# B&R Automation Studio project Code_für_SPS
Automation Studio 4.9

## Configuration Config1

CPU X20CP1382, AutomationRuntime B4.63, Build 4.1.2, Vc V4.62.0

### Task classes (Cpu.sw)
```
Cyclic#4:
  Program1 <- Program1.prg
Binaries: udbdef, mvLoader, FWRules, TCData, ashwac, arconfig, asfw, ashwd, iomap, User, Role, sysconf
Libraries: sys_lib, AsBrStr, runtime, Library, standard, fileio, astime, asieccon
```

### Hardware
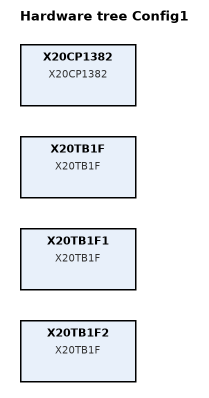
```
X20CP1382 : X20CP1382 v1.14.0.0  [X1 -> X1.SL; X2 -> X2.SL; X3 -> X3.SL]
  Module X1 (Type=X1, Virtual=true, Version=1.14.0.0)
    Connection (Connector=SS1, TargetModule=X20TB1F, TargetConnector=SS)
    Connection (Connector=SL, TargetModule=X20CP1382, TargetConnector=X1)
  Module X2 (Type=X2, Virtual=true, Version=1.14.0.0)
    Connection (Connector=SS1, TargetModule=X20TB1F1, TargetConnector=SS)
    Connection (Connector=SL, TargetModule=X20CP1382, TargetConnector=X2)
  Module X3 (Type=X3, Virtual=true, Version=1.14.0.0)
    Connection (Connector=SS1, TargetModule=X20TB1F2, TargetConnector=SS)
    Connection (Connector=SL, TargetModule=X20CP1382, TargetConnector=X3)
  Connector IF2:
    ActivateDevice = 1
    HostName = x20cp1382
    Mode = Manual
    InternetAddress = 192.168.1.10
    SubnetMask = 255.255.255.0
    InaNodeNumber = 0
  Connector IF3:
    DNAConfiguration = manual
  ConfigurationID = Cocktailmaschine_Config1
  ActivateOpcUa = 1
  OpcUaInformationModels_PV_Version = 1
X20TB1F : X20TB1F v1.0.0.0
X20TB1F1 : X20TB1F v1.0.0.0
X20TB1F2 : X20TB1F v1.0.0.0
```

### IoMap.iom - X20CP1382/IoMap.iom
```iecst
VAR_CONFIG
	::Program1:OutVentil2 AT %QX."X3".DigitalOutput02;
	::Program1:InLichtschranke AT %IX."X2".DigitalInput01;
	::Program1:OutVentil1 AT %QX."X3".DigitalOutput01;
	::Program1:OutVentil3 AT %QX."X3".DigitalOutput03;
	::Program1:OutVentil4 AT %QX."X3".DigitalOutput04;
	::Program1:OutVentil5 AT %QX."X3".DigitalOutput05;
	::Program1:OutVentil6 AT %QX."X3".DigitalOutput06;
	::Program1:OutVentil7 AT %QX."X3".DigitalOutput07;
	::Program1:OutVentil8 AT %QX."X3".DigitalOutput08;
	::Program1:OutPumpe AT %QX."X3".DigitalOutput09;
	::Program1:OutMotorEis AT %QX."X3".DigitalOutput10;
	::Program1:OutLampeGruen AT %QX."X3".DigitalOutput11;
	::Program1:OutLampeRot AT %QX."X3".DigitalOutput12;
	::Program1:InEndlageMotor AT %IX."X2".DigitalInput02;
	::Program1:InEndlageMotor2 AT %IX."X2".DigitalInput03;
	::Program1:InAnalogWaage AT %IW."X1".AnalogInput02;
END_VAR
```

## Logical view

Binary libraries used (declarations not repeated): operator, runtime, astime, AsIecCon, sys_lib, AsBrStr, standard

### Library Logical/Library (IEC)

#### Library.fun - Exported functions and function blocks
```iecst
{REDUND_ERROR} FUNCTION setOutputs : BOOL (*TODO: Add your comment here*) (*$GROUP=User,$CAT=User,$GROUPICON=User.png,$CATICON=User.png*)
	VAR_INPUT
		ventil1 : BOOL;
		ventil2 : BOOL;
		ventil3 : BOOL;
		ventil4 : BOOL;
		ventil5 : BOOL;
		ventil6 : BOOL;
		ventil7 : BOOL;
		ventil8 : BOOL;
		rot : BOOL;
		gruen : BOOL;
		pumpe : BOOL;
		motor : BOOL;
	END_VAR
END_FUNCTION
```

#### setOutputs.ab
```automation-basic
(* TODO: Add your comment here *)
FUNCTION setOutputs
	//OutVentil1 := ventil1;
	//OutVentil2 := ventil2;
	//OutVentil3 := ventil3;
	//OutVentil4 := ventil4;
	//OutVentil5 := ventil5;
	//OutVentil6 := ventil6;
	//OutVentil7 := ventil7;
	//OutVentil8 := ventil8;
	//OutLampeRot := rot;
	//OutLampeGruen := gruen;
	//OutPumpe := pumpe;
	//OutMotorEis := motor;
END_FUNCTION
```

### Package Logical/Libraries - Globale Bibliotheken

- Visualisation Logical/mappView (not shown)

### Program Logical/Program (IEC)

#### Cyclic.st - Cyclic code
```iecst
PROGRAM _CYCLIC
	IF Zustand = TRUE THEN
		//Hier kommt der Befehl zum Anzeigen dert Startseite hin
		OutVentil1 := FALSE;OutVentil2 := FALSE;OutVentil3 := FALSE;OutVentil4 := FALSE;OutVentil5 := FALSE;OutVentil6 := FALSE;
		OutVentil7 := FALSE;OutVentil8 := FALSE;OutLampeRot := FALSE;OutLampeGruen := FALSE;OutPumpe := FALSE;OutMotorEis := FALSE;
		//Wenn Softbutton für die Shots gedrückt wird wird in Zustand 2 gesprungen
		IF ButtonHShot = TRUE THEN
			Zustand := 2;
		END_IF
		//Wenn Softbutton für die Cocktails gedrückt wird wird in Zustand 4 gesprungen
		IF ButtonHCock = TRUE THEN
			Zustand := 4;
		END_IF
	END_IF
END_PROGRAM
```

#### Init.st - Init code
```iecst
PROGRAM _INIT
	Zustand := 1;
END_PROGRAM
```

#### Variables.var - Local variables
```iecst
VAR
	InWiegezelle : INT;
	InLichtschranke : BOOL;
	InEndlageMotor : BOOL;
	ButtonHShot : BOOL; (*Softbutton auf der Hauptseite für die Shots*)
	ButtonHCock : BOOL; (*Softbutton auf der Hauptseite für die Cocktails*)
	ButtonCCock1 : BOOL; (*Softbutton auf der Cocktailseite für den ersten Cocktail*)
	ButtonCCock2 : BOOL; (*Softbutton auf der Cocktailseite für den zweiten Cocktail*)
	ButtonCCock3 : BOOL; (*Softbutton auf der Cocktailseite für den dritten Cocktail*)
	ButtonCCock4 : BOOL; (*Softbutton auf der Cocktailseite für den vierten Cocktail*)
	ButtonCZurueck : BOOL; (*Softbutton auf der Cocktailseite zum zurück auf die Hauptseite navigieren*)
	ButtonSShot1 : BOOL; (*Softbutton auf der Shotseite für den ersten Shot*)
	ButtonSShot2 : BOOL; (*Softbutton auf der Shotseite für den zweiten Shot*)
	ButtonSShot3 : BOOL; (*Softbutton auf der Shotseite für den dritten Shot*)
	ButtonSShot4 : BOOL; (*Softbutton auf der Shotseite für den vierten Shot*)
	ButtonSZurueck : BOOL; (*Softbutton auf der Shotseite zum zurück auf die Hauptseite navigieren*)
	ButtonBEis : BOOL; (*Softbutton auf der Bestellseite Eis-Haken*)
	ButtonBKEis : BOOL; (*Softbutton auf der Bestellseite Eis-Kreuz*)
	ButtonBGross : BOOL; (*Softbutton auf der Bestellseite großer Cocktail*)
	ButtonBKlein : BOOL; (*Softbutton auf der Bestellseite kleiner Cocktail*)
	ButtonBZurueck : BOOL; (*Softbutton auf der Bestellseite zum zurück zu Auswahlseite navigieren*)
	Zustand : SINT; (*Variable für den Zustand*)
	OutVentil1 : BOOL;
	OutVentil2 : BOOL;
	OutVentil3 : BOOL;
	OutVentil4 : BOOL;
	OutVentil5 : BOOL;
	OutVentil6 : BOOL;
	OutVentil7 : BOOL;
	OutVentil8 : BOOL;
	OutLampeRot : BOOL;
	OutLampeGruen : BOOL;
	OutPumpe : BOOL;
	OutMotorEis : BOOL;
END_VAR
```

### Program Logical/Program1 (ANSIC)

#### Variables.var
```iecst
VAR
	ButtonBZurueck : BOOL; (*Navigationbutton auf der Bestellseite zum zurück zu Auswahlseite navigieren*)
	ButtonCStart : BOOL; (*Button zum starten des Cocktails*)
	ButtonCZurueck : BOOL; (*Navigatoinbutton auf der Cocktailseite zum zurück auf die Hauptseite navigieren*)
	ButtonReset : BOOL; (*Button zum zurücksetzen der Variablen*)
	ButtonSStart : BOOL; (*Button zum starten des Shots*)
	ButtonSZurueck : BOOL; (*Navigationbutton auf der Shotseite zum zurück auf die Hauptseite navigieren*)
	Cocktail : USINT;
	CocktailFertig : BOOL;
	Durchgang : USINT;
	EisFertig : BOOL; (*Flag*)
	FlagMotor : BOOL;
	FuellstandB1 : INT; (*Füllstand des 1. Behälters*)
	FuellstandB2 : INT; (*Füllstand des 2. Behälters*)
	FuellstandB3 : INT; (*Füllstand des 3. Behälters*)
	FuellstandB4 : INT; (*Füllstand des 4. Behälters*)
	FuellstandB5 : INT; (*Füllstand des 5. Behälters*)
	FuellstandB6 : INT; (*Füllstand des 6. Behälters*)
	FuellstandB7 : INT; (*Füllstand des 7. Behälters*)
	FuellstandB8 : INT; (*Füllstand des 8. Behälters*)
	Groessenfaktor : REAL;
	InAnalogWaage : INT; (*Werte des Analogeingangs vom Messumformer der Waage*)
	InEndlageMotor : BOOL;
	InEndlageMotor2 : BOOL;
	Motor_Ausgang : BOOL;
	Motor_Hand : BOOL;
	InLichtschranke : BOOL;
	IstGewicht : INT;
	Nachfuellen : BOOL;
	OutLampeGruen : BOOL;
	OutLampeRot : BOOL;
	OutMotorEis : BOOL;
	OutPumpe : BOOL;
	OutVentil1 : BOOL;
	OutVentil2 : BOOL;
	OutVentil3 : BOOL;
	OutVentil4 : BOOL;
	OutVentil5 : BOOL;
	OutVentil6 : BOOL;
	OutVentil7 : BOOL;
	OutVentil8 : BOOL;
	RButtonBEis : BOOL; (*Radiobutton auf der Bestellseite Eis-Haken*)
	RButtonBGross : BOOL; (*Radiobutton auf der Bestellseite großer Cocktail*)
	RButtonBKEis : BOOL; (*Radiobutton auf der Bestellseite Eis-Kreuz*)
	RButtonBKlein : BOOL; (*Radiobutton auf der Bestellseite kleiner Cocktail*)
	RButtonCock1 : BOOL; (*Radiobutton auf der Cocktailseite für den ersten Cocktail*)
	RButtonCock2 : BOOL; (*Radiobutton auf der Cocktailseite für den zweiten Cocktail*)
	RButtonCock3 : BOOL; (*Radiobutton auf der Cocktailseite für den dritten Cocktail*)
	RButtonCock4 : BOOL; (*Radiobutton auf der Cocktailseite für den vierten Cocktail*)
	RButtonCock5 : BOOL; (*Radiobutton auf der Cocktailseite für den Zufallscocktail*)
	RButtonCock6 : BOOL; (*Radiobutton für den richtigen zufälligen Cocktail*)
	RButtonShot1 : BOOL; (*Radiobutton auf der Shotseite für den ersten Shot*)
	RButtonShot2 : BOOL; (*Radiobutton auf der Shotseite für den zweiten Shot*)
	RButtonShot3 : BOOL; (*Radiobutton auf der Shotseite für den dritten Shot*)
	RButtonShot4 : BOOL; (*Radiobutton auf der Shotseite für den vierten Shot*)
	RButtonShot5 : BOOL; (*Radiobutton auf der Shotseite für den Zufallsshot*)
	Reinigung_1 : BOOL;
	Reinigung_2 : BOOL;
	Reinigung_3 : BOOL;
	Reinigung_4 : BOOL;
	Reinigung_5 : BOOL;
	Reinigung_6 : BOOL;
	Reinigung_7 : BOOL;
	Reinigung_8 : BOOL;
	Reinigung_Stopp : BOOL;
	Shot : USINT;
	ShotFertig : BOOL; (*Flag*)
	StartGewicht : INT;
	Zufall : USINT;
	ZufallsZutat : USINT;
	ZufallsZutatG : BOOL;
	ZufallZufall : USINT;
	Zustand : SINT; (*Variable für den Zustand*)
	Zutat1Fertig : BOOL;
	Zutat2Fertig : BOOL;
	Zutat3Fertig : BOOL;
	Zutat4Fertig : BOOL;
END_VAR
```

#### Main.c
```c
#include <bur/plctypes.h>
#ifdef _DEFAULT_INCLUDES
	#include <AsDefault.h>
#endif

_GLOBAL int r_pv;
int rand(void);
void srand(unsigned int seed);
//y = 0,072g/z*x-460g 4cl mit Berücksichtigung des Nachlaufs ca. 530
//1->Tequila 2->Vodka 3->Gin 4->Rum 5->Limettensaft 6->Orangensaft 7->Zitronensaft 8->Tonic Water
//ALTERNATIV 1->Tequila 2->Vodka 3->Gin 4->Rum 5->Limettensaft 6->Orangensaft 7->Ananassaft 8->Tonic Water
void _INIT ProgramInit(void)
{
	Zustand = 1;
	ShotFertig = 1;
	CocktailFertig = 1;
	Cocktail = 0;
	Shot = 0;
	OutLampeGruen = 1;
	Groessenfaktor = 1;
	FuellstandB1 = 9275;
	FuellstandB2 = 9275;
	FuellstandB3 = 9275;
	FuellstandB4 = 9275;
	FuellstandB5 = 9938;
	FuellstandB6 = 53000;
	FuellstandB7 = 53000;
	FuellstandB8 = 53000;
	Nachfuellen = 0;
	srand(12);
	Zufall = 0;
	ZufallsZutatG = 0;
	Durchgang = 1;
	ZufallZufall = 0;
	RButtonCock1 = 1;
	RButtonBKEis = 1;
	RButtonBGross = 1;
	RButtonShot1 = 1;
	FlagMotor = 0;
	Reinigung_1 = 0;
	Reinigung_2 = 0;
	Reinigung_3 = 0;
	Reinigung_4 = 0;
	Reinigung_5 = 0;
	Reinigung_6 = 0;
	Reinigung_7 = 0;
	Reinigung_8 = 0;
	Motor_Hand = 0;
}

void _CYCLIC ProgramCyclic(void)
{
	if(ButtonReset)
	{
		OutVentil1 = 0; OutVentil2 = 0; OutVentil3 = 0; OutVentil4 = 0; OutVentil5 = 0; OutVentil6 = 0;
		OutVentil7 = 0; OutVentil8 = 0; OutLampeRot = 0; OutLampeGruen = 1; OutPumpe = 0; OutMotorEis = 0;
		FuellstandB1 = 9275;
		FuellstandB2 = 9275;
		FuellstandB3 = 9275;
		FuellstandB4 = 9275;
		FuellstandB5 = 9938;
		FuellstandB6 = 53000;
		FuellstandB7 = 53000;
		FuellstandB8 = 53000;
		Zutat1Fertig = 0;
		Zutat2Fertig = 0;
		Zutat3Fertig = 0;
		Zutat4Fertig = 0;
		CocktailFertig = 1;
		ShotFertig = 1;
		IstGewicht = 0;
		StartGewicht = 0;
		Groessenfaktor = 1;
		ButtonReset = 0;
		Zustand = 1;
		Nachfuellen = 0;
		Zufall = 0;
		Durchgang = 1;
		ZufallZufall = 0;
		FlagMotor = 0;
		EisFertig = 0;
		Reinigung_1 = 0;
		Reinigung_2 = 0;
		Reinigung_3 = 0;
		Reinigung_4 = 0;
		Reinigung_5 = 0;
		Reinigung_6 = 0;
		Reinigung_7 = 0;
		Reinigung_8 = 0;
		Motor_Hand = 0;
	}
	// Durchlauf der verschiedenen Zustände
	if(Zustand == 1)
	{
		OutVentil1 = 0; OutVentil2 = 0; OutVentil3 = 0; OutVentil4 = 0; OutVentil5 = 0; OutVentil6 = 0;
		OutVentil7 = 0; OutVentil8 = 0; OutLampeRot = 0; OutLampeGruen = 1; OutPumpe = 0; OutMotorEis = 0;
		CocktailFertig = 1;
		ShotFertig = 1;
	}
	else if(Zustand == 2)
	{
		//Wahl des Shots
		if((!ShotFertig && RButtonShot1 && !Nachfuellen && InLichtschranke) || Zufall == 1)
		{
			OutVentil1 = 1; OutVentil2 = 0; OutVentil3 = 0; OutVentil4 = 0; OutVentil5 = 0; OutVentil6 = 0;
			OutVentil7 = 0; OutVentil8 = 0; OutLampeRot = 1; OutLampeGruen = 0; OutPumpe = 1; OutMotorEis = 0;
			IstGewicht = InAnalogWaage;
			if(IstGewicht - StartGewicht >= 530)
			{
				OutVentil1 = 0; OutVentil2 = 0; OutVentil3 = 0; OutVentil4 = 0; OutVentil5 = 0; OutVentil6 = 0;
				OutVentil7 = 0; OutVentil8 = 0; OutLampeRot = 0; OutLampeGruen = 1; OutPumpe = 0; OutMotorEis = 0;
				ShotFertig = 1;
				FuellstandB1 -= 530;
				Zufall = 0;
			}
			Shot = 1;
		}
		if((!ShotFertig && RButtonShot2 && !Nachfuellen && InLichtschranke) || Zufall == 2)
		{
			OutVentil1 = 0; OutVentil2 = 1; OutVentil3 = 0; OutVentil4 = 0; OutVentil5 = 0; OutVentil6 = 0;
			OutVentil7 = 0; OutVentil8 = 0; OutLampeRot = 1; OutLampeGruen = 0; OutPumpe = 1; OutMotorEis = 0;
			IstGewicht = InAnalogWaage;
			if(IstGewicht - StartGewicht >= 530)
			{
				OutVentil1 = 0; OutVentil2 = 0; OutVentil3 = 0; OutVentil4 = 0; OutVentil5 = 0; OutVentil6 = 0;
				OutVentil7 = 0; OutVentil8 = 0; OutLampeRot = 0; OutLampeGruen = 1; OutPumpe = 0; OutMotorEis = 0;
				ShotFertig = 1;
				FuellstandB2 -= 530;
				Zufall = 0;
			}
			Shot = 2;
		}
		if((!ShotFertig && RButtonShot3 && !Nachfuellen && InLichtschranke) || Zufall == 3)
		{
			OutVentil1 = 0; OutVentil2 = 0; OutVentil3 = 1; OutVentil4 = 0; OutVentil5 = 0; OutVentil6 = 0;
			OutVentil7 = 0; OutVentil8 = 0; OutLampeRot = 1; OutLampeGruen = 0; OutPumpe = 1; OutMotorEis = 0;
			IstGewicht = InAnalogWaage;
			if(IstGewicht - StartGewicht >= 530)
			{
				OutVentil1 = 0; OutVentil2 = 0; OutVentil3 = 0; OutVentil4 = 0; OutVentil5 = 0; OutVentil6 = 0;
				OutVentil7 = 0; OutVentil8 = 0; OutLampeRot = 0; OutLampeGruen = 1; OutPumpe = 0; OutMotorEis = 0;
				ShotFertig = 1;
				FuellstandB3 -= 530;
				Zufall = 0;
			}
			Shot = 3;
		}
		if((!ShotFertig && RButtonShot4 && !Nachfuellen && InLichtschranke) || Zufall == 4)
		{
			OutVentil1 = 0; OutVentil2 = 0; OutVentil3 = 0; OutVentil4 = 1; OutVentil5 = 0; OutVentil6 = 0;
			OutVentil7 = 0; OutVentil8 = 0; OutLampeRot = 1; OutLampeGruen = 0; OutPumpe = 1; OutMotorEis = 0;
			IstGewicht = InAnalogWaage;
			if(IstGewicht - StartGewicht >= 530)
			{
				OutVentil1 = 0; OutVentil2 = 0; OutVentil3 = 0; OutVentil4 = 0; OutVentil5 = 0; OutVentil6 = 0;
				OutVentil7 = 0; OutVentil8 = 0; OutLampeRot = 0; OutLampeGruen = 1; OutPumpe = 0; OutMotorEis = 0;
				ShotFertig = 1;
				FuellstandB4 -= 530;
				Zufall = 0;
			}
			Shot = 4;
		}
		if(!ShotFertig && RButtonShot5 && !Nachfuellen && InLichtschranke && Zufall == 0)
		{
			//Zufallsshot
			Zufall = rand() % 4 + 1;
		}
	}
	else if(Zustand == 3)
	{	//Legspreader
		//Wahl des Cocktails
		if((!CocktailFertig && RButtonCock1 && !Nachfuellen && InLichtschranke) || Zufall == 1)
		{
			Cocktail = 1;
			//Massenanpassungsfaktor bei Größenwahl
			if(RButtonBKlein)
			{
				Groessenfaktor = 0.5;
			}
			if(RButtonBGross)
			{
				Groessenfaktor = 1;
			}
			//Das erste If wird so lange durchlaufen, bis der Motor für das Eis seine Endlage erreicht hat.
			//Oder es wird gar nicht durchlaufen, falls der Benutzer ohne Eis gklickt hat
			if(RButtonBEis && !EisFertig)
			{
				OutVentil1 = 0; OutVentil2 = 0; OutVentil3 = 0; OutVentil4 = 0; OutVentil5 = 0; OutVentil6 = 0;
				OutVentil7 = 0; OutVentil8 = 0; OutLampeRot = 1; OutLampeGruen = 0; OutPumpe = 0; OutMotorEis = 1;
				if(InEndlageMotor2)
				{
					FlagMotor = 1;
				}
				if(InEndlageMotor && FlagMotor)
				{
					OutVentil1 = 0; OutVentil2 = 0; OutVentil3 = 0; OutVentil4 = 0; OutVentil5 = 0; OutVentil6 = 0;
					OutVentil7 = 0; OutVentil8 = 0; OutLampeRot = 1; OutLampeGruen = 0; OutPumpe = 0; OutMotorEis = 0;
					EisFertig = 1;
					FlagMotor = 0;
					StartGewicht = InAnalogWaage;
				}
			}
			else
			{
				//Der If Zweig wird so lange durchlaufen, bis die erste Zutat fertig ist.
				//Anschließend wird nur noch der Else Zweig durchlaufen
				if(!Zutat1Fertig)
				{
					OutVentil1 = 1; OutVentil2 = 0; OutVentil3 = 0; OutVentil4 = 0; OutVentil5 = 0; OutVentil6 = 0;
					OutVentil7 = 0; OutVentil8 = 0; OutLampeRot = 1; OutLampeGruen = 0; OutPumpe = 1; OutMotorEis = 0;
					IstGewicht = InAnalogWaage;
					if(IstGewicht - StartGewicht >= 530 * Groessenfaktor)
					{
						OutVentil1 = 0; OutVentil2 = 0; OutVentil3 = 0; OutVentil4 = 0; OutVentil5 = 0; OutVentil6 = 0;
						OutVentil7 = 0; OutVentil8 = 0; OutLampeRot = 1; OutLampeGruen = 0; OutPumpe = 1; OutMotorEis = 0;
						Zutat1Fertig = 1;
						StartGewicht = InAnalogWaage;
					}
				}
				else
				{
					//Der If Zweig wird so lange durchlaufen, bis die zweite Zutat fertig ist.
					//Anschließend wird nur noch der Else Zweig durchlaufen
					if(!Zutat2Fertig)
					{
						OutVentil1 = 0; OutVentil2 = 0; OutVentil3 = 0; OutVentil4 = 1; OutVentil5 = 0; OutVentil6 = 0;
						OutVentil7 = 0; OutVentil8 = 0; OutLampeRot = 1; OutLampeGruen = 0; OutPumpe = 1; OutMotorEis = 0;
						IstGewicht = InAnalogWaage;
						if(IstGewicht - StartGewicht >= 530 * Groessenfaktor)
						{
							OutVentil1 = 0; OutVentil2 = 0; OutVentil3 = 0; OutVentil4 = 0; OutVentil5 = 0; OutVentil6 = 0;
							OutVentil7 = 0; OutVentil8 = 0; OutLampeRot = 1; OutLampeGruen = 0; OutPumpe = 1; OutMotorEis = 0;
							Zutat2Fertig = 1;
							StartGewicht = InAnalogWaage;
						}
					}
					else
					{
						//Der If Zweig wird so lange durchlaufen, bis die dritte Zutat fertig ist.
						//Anschließend wird nur noch der Else Zweig durchlaufen
						if(!Zutat3Fertig)
						{
							OutVentil1 = 0; OutVentil2 = 0; OutVentil3 = 0; OutVentil4 = 0; OutVentil5 = 0; OutVentil6 = 1;
							OutVentil7 = 0; OutVentil8 = 0; OutLampeRot = 1; OutLampeGruen = 0; OutPumpe = 1; OutMotorEis = 0;
							IstGewicht = InAnalogWaage;
							if(IstGewicht - StartGewicht >= 2000 * Groessenfaktor)
							{
								OutVentil1 = 0; OutVentil2 = 0; OutVentil3 = 0; OutVentil4 = 0; OutVentil5 = 0; OutVentil6 = 0;
								OutVentil7 = 0; OutVentil8 = 0; OutLampeRot = 1; OutLampeGruen = 0; OutPumpe = 1; OutMotorEis = 0;
								Zutat3Fertig = 1;
								StartGewicht = InAnalogWaage;
							}
						}
						else
						{
							//Der If Zweig wird so lange durchlaufen, bis die vierte Zutat fertig ist.
							//Anschließend wird nur noch der Else Zweig durchlaufen
							if(!Zutat4Fertig)
							{
								OutVentil1 = 0; OutVentil2 = 0; OutVentil3 = 0; OutVentil4 = 0; OutVentil5 = 1; OutVentil6 = 0;
								OutVentil7 = 0; OutVentil8 = 0; OutLampeRot = 1; OutLampeGruen = 0; OutPumpe = 1; OutMotorEis = 0;
								IstGewicht = InAnalogWaage;
								if(IstGewicht - StartGewicht >= 265 * Groessenfaktor)
								{
									OutVentil1 = 0; OutVentil2 = 0; OutVentil3 = 0; OutVentil4 = 0; OutVentil5 = 0; OutVentil6 = 0;
									OutVentil7 = 0; OutVentil8 = 0; OutLampeRot = 0; OutLampeGruen = 1; OutPumpe = 0; OutMotorEis = 0;
									Zutat4Fertig = 1;
									CocktailFertig = 1;
									FuellstandB1 -= 530; FuellstandB4 -= 530; FuellstandB6 -= 2000; FuellstandB5 -= 265;
									Zufall = 0;
								}
							}
						}
					}
				}
			}
		}
		if((!CocktailFertig && RButtonCock2 && !Nachfuellen && InLichtschranke) || Zufall == 2)
		{
			Cocktail = 2;
			//Scrumdriver
			//Massenanpassungsfaktor bei Größenwahl
			if(RButtonBKlein)
			{
				Groessenfaktor = 0.5;
			}
			if(RButtonBGross)
			{
				Groessenfaktor = 1;
			}
			//Das erste If wird so lange durchlaufen, bis der Motor für das Eis seine Endlage erreicht hat.
			//Oder es wird gar nicht durchlaufen, falls der Benutzer ohne Eis gklickt hat
			if(RButtonBEis && !EisFertig)
			{
				OutVentil1 = 0; OutVentil2 = 0; OutVentil3 = 0; OutVentil4 = 0; OutVentil5 = 0; OutVentil6 = 0;
				OutVentil7 = 0; OutVentil8 = 0; OutLampeRot = 1; OutLampeGruen = 0; OutPumpe = 0; OutMotorEis = 1;
				if(InEndlageMotor2)
				{
					FlagMotor = 1;
				}
				if(InEndlageMotor && FlagMotor)
				{
					OutVentil1 = 0; OutVentil2 = 0; OutVentil3 = 0; OutVentil4 = 0; OutVentil5 = 0; OutVentil6 = 0;
					OutVentil7 = 0; OutVentil8 = 0; OutLampeRot = 1; OutLampeGruen = 0; OutPumpe = 0; OutMotorEis = 0;
					EisFertig = 1;
					FlagMotor = 0;
					StartGewicht = InAnalogWaage;
				}
			}
			else
			{
				//Der If Zweig wird so lange durchlaufen, bis die erste Zutat fertig ist.
				//Anschließend wird nur noch der Else Zweig durchlaufen
				if(!Zutat1Fertig)
				{
					OutVentil1 = 0; OutVentil2 = 0; OutVentil3 = 1; OutVentil4 = 0; OutVentil5 = 0; OutVentil6 = 0;
					OutVentil7 = 0; OutVentil8 = 0; OutLampeRot = 1; OutLampeGruen = 0; OutPumpe = 1; OutMotorEis = 0;
					IstGewicht = InAnalogWaage;
					if(IstGewicht - StartGewicht >= 660 * Groessenfaktor)
					{
						OutVentil1 = 0; OutVentil2 = 0; OutVentil3 = 0; OutVentil4 = 0; OutVentil5 = 0; OutVentil6 = 0;
						OutVentil7 = 0; OutVentil8 = 0; OutLampeRot = 1; OutLampeGruen = 0; OutPumpe = 1; OutMotorEis = 0;
						Zutat1Fertig = 1;
						StartGewicht = InAnalogWaage;
					}
				}
				else
				{
					//Der If Zweig wird so lange durchlaufen, bis die zweite Zutat fertig ist.
					//Anschließend wird nur noch der Else Zweig durchlaufen
					if(!Zutat2Fertig)
					{
						OutVentil1 = 0; OutVentil2 = 0; OutVentil3 = 0; OutVentil4 = 0; OutVentil5 = 0; OutVentil6 = 0;
						OutVentil7 = 0; OutVentil8 = 1; OutLampeRot = 1; OutLampeGruen = 0; OutPumpe = 1; OutMotorEis = 0;
						IstGewicht = InAnalogWaage;
						if(IstGewicht - StartGewicht >= 2385 * Groessenfaktor)
						{
							OutVentil1 = 0; OutVentil2 = 0; OutVentil3 = 0; OutVentil4 = 0; OutVentil5 = 0; OutVentil6 = 0;
							OutVentil7 = 0; OutVentil8 = 0; OutLampeRot = 1; OutLampeGruen = 0; OutPumpe = 1; OutMotorEis = 0;
							Zutat2Fertig = 1;
							StartGewicht = InAnalogWaage;
						}
					}
					else
					{
						//Der If Zweig wird so lange durchlaufen, bis die dritte Zutat fertig ist.
						//Anschließend wird nur noch der Else Zweig durchlaufen
						if(!Zutat3Fertig)
						{
							OutVentil1 = 0; OutVentil2 = 0; OutVentil3 = 0; OutVentil4 = 0; OutVentil5 = 1; OutVentil6 = 0;
							OutVentil7 = 0; OutVentil8 = 0; OutLampeRot = 1; OutLampeGruen = 0; OutPumpe = 1; OutMotorEis = 0;
							IstGewicht = InAnalogWaage;
							if(IstGewicht - StartGewicht >= 265 * Groessenfaktor)
							{
								OutVentil1 = 0; OutVentil2 = 0; OutVentil3 = 0; OutVentil4 = 0; OutVentil5 = 0; OutVentil6 = 0;
								OutVentil7 = 0; OutVentil8 = 0; OutLampeRot = 0; OutLampeGruen = 1; OutPumpe = 0; OutMotorEis = 0;
								Zutat3Fertig = 1;
								CocktailFertig = 1;
								FuellstandB3 -= 660; FuellstandB8 -= 2385; FuellstandB2 -= 265;
								Zufall = 0;
							}
						}
					}
				}
			}
		}
		if((!CocktailFertig && RButtonCock3 && !Nachfuellen && InLichtschranke) || Zufall == 3)
		{
			Cocktail = 3;
			//Gentle Ben
			//Massenanpassungsfaktor bei Größenwahl
			if(RButtonBKlein)
			{
				Groessenfaktor = 0.5;
			}
			if(RButtonBGross)
			{
				Groessenfaktor = 1;
			}
			//Das erste If wird so lange durchlaufen, bis der Motor für das Eis seine Endlage erreicht hat.
			//Oder es wird gar nicht durchlaufen, falls der Benutzer ohne Eis gklickt hat
			if(RButtonBEis && !EisFertig)
			{
				OutVentil1 = 0; OutVentil2 = 0; OutVentil3 = 0; OutVentil4 = 0; OutVentil5 = 0; OutVentil6 = 0;
				OutVentil7 = 0; OutVentil8 = 0; OutLampeRot = 1; OutLampeGruen = 0; OutPumpe = 0; OutMotorEis = 1;
				if(InEndlageMotor2)
				{
					FlagMotor = 1;
				}
				if(InEndlageMotor && FlagMotor)
				{
					OutVentil1 = 0; OutVentil2 = 0; OutVentil3 = 0; OutVentil4 = 0; OutVentil5 = 0; OutVentil6 = 0;
					OutVentil7 = 0; OutVentil8 = 0; OutLampeRot = 1; OutLampeGruen = 0; OutPumpe = 0; OutMotorEis = 0;
					EisFertig = 1;
					FlagMotor = 0;
					StartGewicht = InAnalogWaage;
				}
			}
			else
			{
				//Der If Zweig wird so lange durchlaufen, bis die erste Zutat fertig ist.
				//Anschließend wird nur noch der Else Zweig durchlaufen
				if(!Zutat1Fertig)
				{
					OutVentil1 = 0; OutVentil2 = 0; OutVentil3 = 0; OutVentil4 = 1; OutVentil5 = 0; OutVentil6 = 0;
					OutVentil7 = 0; OutVentil8 = 0; OutLampeRot = 1; OutLampeGruen = 0; OutPumpe = 1; OutMotorEis = 0;
					IstGewicht = InAnalogWaage;
					if(IstGewicht - StartGewicht >= 660 * Groessenfaktor)
					{
						OutVentil1 = 0; OutVentil2 = 0; OutVentil3 = 0; OutVentil4 = 0; OutVentil5 = 0; OutVentil6 = 0;
						OutVentil7 = 0; OutVentil8 = 0; OutLampeRot = 1; OutLampeGruen = 0; OutPumpe = 1; OutMotorEis = 0;
						Zutat1Fertig = 1;
						StartGewicht = InAnalogWaage;
					}
				}
				else
				{
					//Der If Zweig wird so lange durchlaufen, bis die zweite Zutat fertig ist.
					//Anschließend wird nur noch der Else Zweig durchlaufen
					if(!Zutat2Fertig)
					{
						OutVentil1 = 0; OutVentil2 = 0; OutVentil3 = 0; OutVentil4 = 0; OutVentil5 = 1; OutVentil6 = 0;
						OutVentil7 = 0; OutVentil8 = 0; OutLampeRot = 1; OutLampeGruen = 0; OutPumpe = 1; OutMotorEis = 0;
						IstGewicht = InAnalogWaage;
						if(IstGewicht - StartGewicht >= 265 * Groessenfaktor)
						{
							OutVentil1 = 0; OutVentil2 = 0; OutVentil3 = 0; OutVentil4 = 0; OutVentil5 = 0; OutVentil6 = 0;
							OutVentil7 = 0; OutVentil8 = 0; OutLampeRot = 1; OutLampeGruen = 0; OutPumpe = 1; OutMotorEis = 0;
							Zutat2Fertig = 1;
							StartGewicht = InAnalogWaage;
						}
					}
					else
					{
						//Der If Zweig wird so lange durchlaufen, bis die dritte Zutat fertig ist.
						//Anschließend wird nur noch der Else Zweig durchlaufen
						if(!Zutat3Fertig)
						{
							OutVentil1 = 0; OutVentil2 = 0; OutVentil3 = 0; OutVentil4 = 0; OutVentil5 = 0; OutVentil6 = 0;
							OutVentil7 = 1; OutVentil8 = 0; OutLampeRot = 1; OutLampeGruen = 0; OutPumpe = 1; OutMotorEis = 0;
							IstGewicht = InAnalogWaage;
							if(IstGewicht - StartGewicht >= 1722 * Groessenfaktor)
							{
								OutVentil1 = 0; OutVentil2 = 0; OutVentil3 = 0; OutVentil4 = 0; OutVentil5 = 0; OutVentil6 = 0;
								OutVentil7 = 0; OutVentil8 = 0; OutLampeRot = 1; OutLampeGruen = 0; OutPumpe = 1; OutMotorEis = 0;
								Zutat3Fertig = 1;
								StartGewicht = InAnalogWaage;
							}
						}
						else
						{
							//Der If Zweig wird so lange durchlaufen, bis die vierte Zutat fertig ist.
							//Anschließend wird nur noch der Else Zweig durchlaufen
							if(!Zutat4Fertig)
							{
								OutVentil1 = 0; OutVentil2 = 0; OutVentil3 = 0; OutVentil4 = 0; OutVentil5 = 0; OutVentil6 = 0;
								OutVentil7 = 0; OutVentil8 = 1; OutLampeRot = 1; OutLampeGruen = 0; OutPumpe = 1; OutMotorEis = 0;
								IstGewicht = InAnalogWaage;
								if(IstGewicht - StartGewicht >= 660 * Groessenfaktor)
								{
									OutVentil1 = 0; OutVentil2 = 0; OutVentil3 = 0; OutVentil4 = 0; OutVentil5 = 0; OutVentil6 = 0;
									OutVentil7 = 0; OutVentil8 = 0; OutLampeRot = 0; OutLampeGruen = 1; OutPumpe = 0; OutMotorEis = 0;
									Zutat4Fertig = 1;
									CocktailFertig = 1;
									FuellstandB4 -= 660; FuellstandB5 -= 265; FuellstandB7 -= 1722; FuellstandB8 -= 660;
									Zufall = 0;
								}
							}
						}
					}
				}
			}
		}
		if((!CocktailFertig && RButtonCock4 && !Nachfuellen && InLichtschranke) || Zufall == 4)
		{
			Cocktail = 4;
			//Carl Oehl
			//Massenanpassungsfaktor bei Größenwahl
			if(RButtonBKlein)
			{
				Groessenfaktor = 0.5;
			}
			if(RButtonBGross)
			{
				Groessenfaktor = 1;
			}
			//Das erste If wird so lange durchlaufen, bis der Motor für das Eis seine Endlage erreicht hat.
			//Oder es wird gar nicht durchlaufen, falls der Benutzer ohne Eis gklickt hat
			if(RButtonBEis && !EisFertig)
			{
				OutVentil1 = 0; OutVentil2 = 0; OutVentil3 = 0; OutVentil4 = 0; OutVentil5 = 0; OutVentil6 = 0;
				OutVentil7 = 0; OutVentil8 = 0; OutLampeRot = 1; OutLampeGruen = 0; OutPumpe = 0; OutMotorEis = 1;
				if(InEndlageMotor2)
				{
					FlagMotor = 1;
				}
				if(InEndlageMotor && FlagMotor)
				{
					OutVentil1 = 0; OutVentil2 = 0; OutVentil3 = 0; OutVentil4 = 0; OutVentil5 = 0; OutVentil6 = 0;
					OutVentil7 = 0; OutVentil8 = 0; OutLampeRot = 1; OutLampeGruen = 0; OutPumpe = 0; OutMotorEis = 0;
					EisFertig = 1;
					FlagMotor = 0;
					StartGewicht = InAnalogWaage;
				}
			}
			else
			{
				//Der If Zweig wird so lange durchlaufen, bis die erste Zutat fertig ist.
				//Anschließend wird nur noch der Else Zweig durchlaufen
				if(!Zutat1Fertig)
				{
					OutVentil1 = 0; OutVentil2 = 1; OutVentil3 = 0; OutVentil4 = 0; OutVentil5 = 0; OutVentil6 = 0;
					OutVentil7 = 0; OutVentil8 = 0; OutLampeRot = 1; OutLampeGruen = 0; OutPumpe = 1; OutMotorEis = 0;
					IstGewicht = InAnalogWaage;
					if(IstGewicht - StartGewicht >= 265 * Groessenfaktor)
					{
						OutVentil1 = 0; OutVentil2 = 0; OutVentil3 = 0; OutVentil4 = 0; OutVentil5 = 0; OutVentil6 = 0;
						OutVentil7 = 0; OutVentil8 = 0; OutLampeRot = 1; OutLampeGruen = 0; OutPumpe = 1; OutMotorEis = 0;
						Zutat1Fertig = 1;
						StartGewicht = InAnalogWaage;
					}
				}
				else
				{
					//Der If Zweig wird so lange durchlaufen, bis die zweite Zutat fertig ist.
					//Anschließend wird nur noch der Else Zweig durchlaufen
					if(!Zutat2Fertig)
					{
						OutVentil1 = 0; OutVentil2 = 0; OutVentil3 = 0; OutVentil4 = 0; OutVentil5 = 0; OutVentil6 = 1;
						OutVentil7 = 0; OutVentil8 = 0; OutLampeRot = 1; OutLampeGruen = 0; OutPumpe = 1; OutMotorEis = 0;
						IstGewicht = InAnalogWaage;
						if(IstGewicht - StartGewicht >= 1590 * Groessenfaktor)
						{
							OutVentil1 = 0; OutVentil2 = 0; OutVentil3 = 0; OutVentil4 = 0; OutVentil5 = 0; OutVentil6 = 0;
							OutVentil7 = 0; OutVentil8 = 0; OutLampeRot = 1; OutLampeGruen = 0; OutPumpe = 1; OutMotorEis = 0;
							Zutat2Fertig = 1;
							StartGewicht = InAnalogWaage;
						}
					}
					else
					{
						//Der If Zweig wird so lange durchlaufen, bis die dritte Zutat fertig ist.
						//Anschließend wird nur noch der Else Zweig durchlaufen
						if(!Zutat3Fertig)
						{
							OutVentil1 = 0; OutVentil2 = 0; OutVentil3 = 0; OutVentil4 = 0; OutVentil5 = 0; OutVentil6 = 0;
							OutVentil7 = 1; OutVentil8 = 0; OutLampeRot = 1; OutLampeGruen = 0; OutPumpe = 1; OutMotorEis = 0;
							IstGewicht = InAnalogWaage;
							if(IstGewicht - StartGewicht >= 1200 * Groessenfaktor)
							{
								OutVentil1 = 0; OutVentil2 = 0; OutVentil3 = 0; OutVentil4 = 0; OutVentil5 = 0; OutVentil6 = 0;
								OutVentil7 = 0; OutVentil8 = 0; OutLampeRot = 1; OutLampeGruen = 0; OutPumpe = 1; OutMotorEis = 0;
								Zutat3Fertig = 1;
								StartGewicht = InAnalogWaage;
							}
						}
						else
						{
							//Der If Zweig wird so lange durchlaufen, bis die vierte Zutat fertig ist.
							//Anschließend wird nur noch der Else Zweig durchlaufen
							if(!Zutat4Fertig)
							{
								OutVentil1 = 1; OutVentil2 = 0; OutVentil3 = 0; OutVentil4 = 0; OutVentil5 = 0; OutVentil6 = 0;
								OutVentil7 = 0; OutVentil8 = 0; OutLampeRot = 1; OutLampeGruen = 0; OutPumpe = 1; OutMotorEis = 0;
								IstGewicht = InAnalogWaage;
								if(IstGewicht - StartGewicht >= 265 * Groessenfaktor)
								{
									OutVentil1 = 0; OutVentil2 = 0; OutVentil3 = 0; OutVentil4 = 0; OutVentil5 = 0; OutVentil6 = 0;
									OutVentil7 = 0; OutVentil8 = 0; OutLampeRot = 0; OutLampeGruen = 1; OutPumpe = 0; OutMotorEis = 0;
									Zutat4Fertig = 1;
									CocktailFertig = 1;
									FuellstandB2 -= 400; FuellstandB6 -= 1330; FuellstandB7 -= 1200; FuellstandB1 -= 400;
									Zufall = 0;
								}
							}
						}
					}
				}
			}
		}
		if(!CocktailFertig && RButtonCock5 && !Nachfuellen && InLichtschranke && Zufall == 0)
		{
			//Zufälliger Cocktail
			Zufall = rand() % 4 + 1;
		}
		if(!CocktailFertig && RButtonCock6 && !Nachfuellen && InLichtschranke)
		{
			//Richtig zufälliger Cocktail
			Cocktail = 6;
			//Massenanpassungsfaktor bei Größenwahl
			if(RButtonBKlein)
			{
				Groessenfaktor = 0.5;
			}
			if(RButtonBGross)
			{
				Groessenfaktor = 1;
			}
			//Das erste If wird so lange durchlaufen, bis der Motor für das Eis seine Endlage erreicht hat.
			//Oder es wird gar nicht durchlaufen, falls der Benutzer ohne Eis gklickt hat
			if(RButtonBEis && !EisFertig)
			{
				OutVentil1 = 0; OutVentil2 = 0; OutVentil3 = 0; OutVentil4 = 0; OutVentil5 = 0; OutVentil6 = 0;
				OutVentil7 = 0; OutVentil8 = 0; OutLampeRot = 1; OutLampeGruen = 0; OutPumpe = 0; OutMotorEis = 1;
				if(InEndlageMotor2)
				{
					FlagMotor = 1;
				}
				if(InEndlageMotor && FlagMotor)
				{
					OutVentil1 = 0; OutVentil2 = 0; OutVentil3 = 0; OutVentil4 = 0; OutVentil5 = 0; OutVentil6 = 0;
					OutVentil7 = 0; OutVentil8 = 0; OutLampeRot = 1; OutLampeGruen = 0; OutPumpe = 0; OutMotorEis = 0;
					EisFertig = 1;
					FlagMotor = 0;
					StartGewicht = InAnalogWaage;
				}
			}
			else
			{
				if(ZufallZufall == 0)
				{
					ZufallZufall = rand() % 8 + 1;
				}
				else
				{
					switch(ZufallZufall)
					{
						case 1:
							OutVentil1 = 1; OutVentil2 = 0; OutVentil3 = 0; OutVentil4 = 0; OutVentil5 = 0; OutVentil6 = 0;
							OutVentil7 = 0; OutVentil8 = 0; OutLampeRot = 1; OutLampeGruen = 0; OutPumpe = 1; OutMotorEis = 0;
							break;
						case 2:
							OutVentil1 = 0; OutVentil2 = 1; OutVentil3 = 0; OutVentil4 = 0; OutVentil5 = 0; OutVentil6 = 0;
							OutVentil7 = 0; OutVentil8 = 0; OutLampeRot = 1; OutLampeGruen = 0; OutPumpe = 1; OutMotorEis = 0;
							break;
						case 3:
							OutVentil1 = 0; OutVentil2 = 0; OutVentil3 = 1; OutVentil4 = 0; OutVentil5 = 0; OutVentil6 = 0;
							OutVentil7 = 0; OutVentil8 = 0; OutLampeRot = 1; OutLampeGruen = 0; OutPumpe = 1; OutMotorEis = 0;
							break;
						case 4:
							OutVentil1 = 0; OutVentil2 = 0; OutVentil3 = 0; OutVentil4 = 1; OutVentil5 = 0; OutVentil6 = 0;
							OutVentil7 = 0; OutVentil8 = 0; OutLampeRot = 1; OutLampeGruen = 0; OutPumpe = 1; OutMotorEis = 0;
							break;
						case 5:
							OutVentil1 = 0; OutVentil2 = 0; OutVentil3 = 0; OutVentil4 = 0; OutVentil5 = 1; OutVentil6 = 0;
							OutVentil7 = 0; OutVentil8 = 0; OutLampeRot = 1; OutLampeGruen = 0; OutPumpe = 1; OutMotorEis = 0;
							break;
						case 6:
							OutVentil1 = 0; OutVentil2 = 0; OutVentil3 = 0; OutVentil4 = 0; OutVentil5 = 0; OutVentil6 = 1;
							OutVentil7 = 0; OutVentil8 = 0; OutLampeRot = 1; OutLampeGruen = 0; OutPumpe = 1; OutMotorEis = 0;
							break;
						case 7:
							OutVentil1 = 0; OutVentil2 = 0; OutVentil3 = 0; OutVentil4 = 0; OutVentil5 = 0; OutVentil6 = 0;
							OutVentil7 = 1; OutVentil8 = 0; OutLampeRot = 1; OutLampeGruen = 0; OutPumpe = 1; OutMotorEis = 0;
							break;
						case 8:
							OutVentil1 = 0; OutVentil2 = 0; OutVentil3 = 0; OutVentil4 = 0; OutVentil5 = 0; OutVentil6 = 0;
							OutVentil7 = 0; OutVentil8 = 1; OutLampeRot = 1; OutLampeGruen = 0; OutPumpe = 1; OutMotorEis = 0;
							break;
						default:
							break;
					}
				}
				IstGewicht = InAnalogWaage;
				if(IstGewicht - StartGewicht >= 1000 * Groessenfaktor)
				{
					OutVentil1 = 0; OutVentil2 = 0; OutVentil3 = 0; OutVentil4 = 0; OutVentil5 = 0; OutVentil6 = 0;
					OutVentil7 = 0; OutVentil8 = 0; OutLampeRot = 1; OutLampeGruen = 0; OutPumpe = 1; OutMotorEis = 0;
					StartGewicht = InAnalogWaage;
					switch(ZufallZufall)
					{
						case 1: FuellstandB1-=1000*Groessenfaktor;break;
						case 2: FuellstandB2-=1000*Groessenfaktor;break;
						case 3: FuellstandB3-=1000*Groessenfaktor;break;
						case 4: FuellstandB4-=1000*Groessenfaktor;break;
						case 5: FuellstandB5-=1000*Groessenfaktor;break;
						case 6: FuellstandB6-=1000*Groessenfaktor;break;
						case 7: FuellstandB7-=1000*Groessenfaktor;break;
						case 8: FuellstandB8-=1000*Groessenfaktor;break;
					}
					ZufallZufall = 0;
					Durchgang++;
				}
				if(Durchgang == 5)
				{
					CocktailFertig = 1;
					OutVentil1 = 0; OutVentil2 = 0; OutVentil3 = 0; OutVentil4 = 0; OutVentil5 = 0; OutVentil6 = 0;
					OutVentil7 = 0; OutVentil8 = 0; OutLampeRot = 0; OutLampeGruen = 1; OutPumpe = 0; OutMotorEis = 0;
					Durchgang = 1;
				}
			}
		}
	}

	//Zustandswechsel
	if(ButtonSStart && ShotFertig && !Nachfuellen && InLichtschranke)
	{
		Zustand = 2;
		ShotFertig = 0;
		StartGewicht = InAnalogWaage;
		ButtonSStart = 0;
	}
	if(ButtonCStart && CocktailFertig && !Nachfuellen && InLichtschranke)
	{
		Zustand = 3;
		CocktailFertig = 0;
		StartGewicht = InAnalogWaage;
		ButtonCStart = 0;
		Zutat1Fertig = 0;
		Zutat2Fertig = 0;
		Zutat3Fertig = 0;
		Zutat4Fertig = 0;
		EisFertig = 0;
	}
	//Abziehen der Massen
	if(FuellstandB1 <= 1000 || FuellstandB3 <= 1000 || FuellstandB3 <= 1000 || FuellstandB4 <= 1000 ||
		FuellstandB5 <= 1000 || FuellstandB6 <= 3000 || FuellstandB7 <= 3000 || FuellstandB8 <= 3000)
	{
		Nachfuellen = 1;
	}

	if(Reinigung_1){
		OutVentil1 = 1; OutVentil2 = 0; OutVentil3 = 0; OutVentil4 = 0; OutVentil5 = 0; OutVentil6 = 0;
		OutVentil7 = 0; OutVentil8 = 0; OutLampeRot = 1; OutLampeGruen = 0; OutPumpe = 1; OutMotorEis = 0;
	}
	if(Reinigung_2){
		OutVentil1 = 0; OutVentil2 = 1; OutVentil3 = 0; OutVentil4 = 0; OutVentil5 = 0; OutVentil6 = 0;
		OutVentil7 = 0; OutVentil8 = 0; OutLampeRot = 1; OutLampeGruen = 0; OutPumpe = 1; OutMotorEis = 0;
	}
	if(Reinigung_3){
		OutVentil1 = 0; OutVentil2 = 0; OutVentil3 = 1; OutVentil4 = 0; OutVentil5 = 0; OutVentil6 = 0;
		OutVentil7 = 0; OutVentil8 = 0; OutLampeRot = 1; OutLampeGruen = 0; OutPumpe = 1; OutMotorEis = 0;
	}
	if(Reinigung_4){
		OutVentil1 = 0; OutVentil2 = 0; OutVentil3 = 0; OutVentil4 = 1; OutVentil5 = 0; OutVentil6 = 0;
		OutVentil7 = 0; OutVentil8 = 0; OutLampeRot = 1; OutLampeGruen = 0; OutPumpe = 1; OutMotorEis = 0;
	}
	if(Reinigung_5){
		OutVentil1 = 0; OutVentil2 = 0; OutVentil3 = 0; OutVentil4 = 0; OutVentil5 = 1; OutVentil6 = 0;
		OutVentil7 = 0; OutVentil8 = 0; OutLampeRot = 1; OutLampeGruen = 0; OutPumpe = 1; OutMotorEis = 0;
	}
	if(Reinigung_6){
		OutVentil1 = 0; OutVentil2 = 0; OutVentil3 = 0; OutVentil4 = 0; OutVentil5 = 0; OutVentil6 = 1;
		OutVentil7 = 0; OutVentil8 = 0; OutLampeRot = 1; OutLampeGruen = 0; OutPumpe = 1; OutMotorEis = 0;
	}
	if(Reinigung_7){
		OutVentil1 = 0; OutVentil2 = 0; OutVentil3 = 0; OutVentil4 = 0; OutVentil5 = 0; OutVentil6 = 0;
		OutVentil7 = 1; OutVentil8 = 0; OutLampeRot = 1; OutLampeGruen = 0; OutPumpe = 1; OutMotorEis = 0;
	}
	if(Reinigung_8){
		OutVentil1 = 0; OutVentil2 = 0; OutVentil3 = 0; OutVentil4 = 0; OutVentil5 = 0; OutVentil6 = 0;
		OutVentil7 = 0; OutVentil8 = 1; OutLampeRot = 1; OutLampeGruen = 0; OutPumpe = 1; OutMotorEis = 0;
	}
	if(Motor_Hand){
		OutVentil1 = 0; OutVentil2 = 0; OutVentil3 = 0; OutVentil4 = 0; OutVentil5 = 0; OutVentil6 = 0;
		OutVentil7 = 0; OutVentil8 = 0; OutLampeRot = 1; OutLampeGruen = 0; OutPumpe = 0; OutMotorEis = 1;
	}
	if(Motor_Ausgang){
		if(InEndlageMotor){
			OutVentil1 = 0; OutVentil2 = 0; OutVentil3 = 0; OutVentil4 = 0; OutVentil5 = 0; OutVentil6 = 0;
			OutVentil7 = 0; OutVentil8 = 0; OutLampeRot = 0; OutLampeGruen = 1; OutPumpe = 0; OutMotorEis = 0;
			Motor_Ausgang = 0;
		}
		else{
			OutVentil1 = 0; OutVentil2 = 0; OutVentil3 = 0; OutVentil4 = 0; OutVentil5 = 0; OutVentil6 = 0;
			OutVentil7 = 0; OutVentil8 = 0; OutLampeRot = 1; OutLampeGruen = 0; OutPumpe = 0; OutMotorEis = 1;
		}
	}
	if(Reinigung_Stopp){
		OutVentil1 = 0; OutVentil2 = 0; OutVentil3 = 0; OutVentil4 = 0; OutVentil5 = 0; OutVentil6 = 0;
		OutVentil7 = 0; OutVentil8 = 0; OutLampeRot = 0; OutLampeGruen = 1; OutPumpe = 0; OutMotorEis = 0;
		Reinigung_1 = 0;
		Reinigung_2 = 0;
		Reinigung_3 = 0;
		Reinigung_4 = 0;
		Reinigung_5 = 0;
		Reinigung_6 = 0;
		Reinigung_7 = 0;
		Reinigung_8 = 0;
		Motor_Hand = 0;
	}
	ButtonSStart = 0;
	ButtonCStart = 0;
	Reinigung_Stopp = 0;
}

void _EXIT ProgramExit(void)
{

}
```

Listed in the project but not available here: Logical/Global.typ, Logical/Global.var, Logical/Library/Types.typ, Logical/Library/Constants.var, Logical/Program/Exit.st, Logical/Program/Types.typ
